// TwinCAT 3 PLC project TRAJ_ADS_SERVER
// ProgramVersion: 3.1.4020.4
// libraries:
//   Tc2_ControllerToolbox, * (Beckhoff Automation GmbH)
//   Tc2_Standard, * (Beckhoff Automation GmbH)
//   Tc2_System, * (Beckhoff Automation GmbH)
//   Tc3_Interfaces, * (Beckhoff Automation GmbH)
//   Tc3_Module, * (Beckhoff Automation GmbH)
// project tree:
//   DUTs/ ROBOT_STATUS.TcDUT (not stored), TRAJECTORY.TcDUT, TRAJ_POINT.TcDUT
//   GVLs/ CONST.TcGVL (not stored)
//   / PlcTask.TcTTO
//   POUs/ MAIN.TcPOU
// real-time tasks:
//   TASK PlcTask: cycle T#1ms, priority 6, ADS port 350
// motion (NC):
//   TASK NC-Task 1 SAF: cycle T#2ms, priority 4, ADS port 501
//   TASK NC-Task 1 SVB: cycle T#10ms, priority 8, ADS port 511
//   AXIS Axis 1 (id 1)
//     OtherSettings: AllowMotionCmdToSlave=true
//     encoder EncType=19
//       EncPara: MaxCount=#xffffffff
//     drive DrvType=16
//       DrvPara: MaxCount=#xffffffff, DriveControlDWord=#x00000100
//         Analog: ScaleFactorActTorque=0.1
//         TimeComp: TaskDelayCycles=1
//     controller CtrType=1
//       CtrPara: PriorControlFactor=1
//         Observer: BandWidth=20
// I/O:
//   DEVICE MY_MOTOR (EtherCAT), AmsNetId 192.168.6.90.3.1
//     Drive 1 (SanyoDenki RS2 EtherCAT) [R ADVANCED MODEL with EtherCAT(P0002813G01)]
// variable links:
//   NC-Task 1 SAF/Axes/Axis 1 <-> MY_MOTOR (EtherCAT)/Drive 1 (SanyoDenki RS2 EtherCAT)
//     Drive/Inputs/In/nDataIn1 <-> Inputs/Following error actualvalue
//     Drive/Inputs/In/nDcOutputTime <-> InfoData/DcOutputShift
//     Drive/Inputs/In/nState1 <-> Inputs/Status word
//     Drive/Inputs/In/nState2 <-> Inputs/Status word @bit 8
//     Drive/Inputs/In/nState4 @bit 1 <-> WcState/InputToggle
//     Drive/Inputs/In/nState4 <-> WcState/WcState
//     Drive/Outputs/Out/nDataOut1 <-> Outputs/Target position
//     Drive/Outputs/Out/nDataOut2 <-> Outputs/Target velocity
//     Enc/Inputs/In/nDataIn3 <-> Inputs/Touch probe position 1 positive value
//     Enc/Inputs/In/nDataIn4 <-> Inputs/Touch probe position 1 negative value
//     Enc/Inputs/In/nDcInputTime <-> InfoData/DcInputShift
//     Enc/Inputs/In/nState4 @bit 1 <-> WcState/InputToggle
//     Enc/Inputs/In/nState4 <-> WcState/WcState
//     Enc/Inputs/In/nState5 <-> Inputs/Touch probe status
//     Enc/Inputs/In/nState6 <-> Inputs/Touch probe status @bit 8
//     Enc/Outputs/Out/nCtrl5 <-> Outputs/Touch probe function
//     Enc/Outputs/Out/nCtrl6 <-> Outputs/Touch probe function @bit 8
//   TRAJ_ADS_SERVER/TRAJ_ADS_SERVER Instance <-> MY_MOTOR (EtherCAT)/Drive 1 (SanyoDenki RS2 EtherCAT)
//     PlcTask Inputs/MAIN.posAct <-> Inputs/Position actual value
//     PlcTask Inputs/MAIN.torAct <-> Inputs/Torque actual value
//     PlcTask Inputs/MAIN.velAct <-> Inputs/Velocity actual value
//     PlcTask Outputs/MAIN.torSet <-> Outputs/Target torque

CONFIGURATION TRAJ_ADS_SERVER
    RESOURCE PLC ON TwinCAT3
        TASK PlcTask(INTERVAL := T#10ms, PRIORITY := 6);
        PROGRAM MAIN WITH PlcTask : MAIN;
    END_RESOURCE
END_CONFIGURATION

// ---- DUTs/TRAJECTORY.TcDUT
TYPE TRAJECTORY :
STRUCT
		size     	  :UINT:=0;                          //轨迹点的数目
		//points        :ARRAY[0..100] OF this_point;      //要执行的一系列轨迹点  
END_STRUCT
END_TYPE

// ---- DUTs/TRAJ_POINT.TcDUT
TYPE TRAJ_POINT :
STRUCT
	joints    : ARRAY [0..6] OF REAL;              //关节的位置数据(7关节)
END_STRUCT
END_TYPE

// ---- POUs/MAIN.TcPOU
PROGRAM MAIN

VAR CONSTANT
	TRAJ_CMD_STOP: 	BYTE :=  0;//停止
	TRAJ_CMD_NEW:   BYTE :=  1;//读入轨迹
	TRAJ_CMD_START: BYTE :=  2;//开始运动
	PULSE_NUM:LREAL:=131072; //编码器脉冲长度
	CYCLE_TICK:BYTE:=1;//周期1us
END_VAR

VAR
	//ADS变量
	traj_cmd                :BYTE:=TRAJ_CMD_STOP; //命令
	traj_size               :UINT:=10;       					//轨迹点的个数
    points        			:ARRAY[0..100] OF TRAJ_POINT;      //要执行的一系列轨迹点 
	joints    : ARRAY [0..6] OF REAL;                  //关节位置数组
	traj_point :TRAJ_POINT;    			   //执行的轨迹点
	last_point :TRAJ_POINT;    			   //执行的轨迹点
	step  :UINT:=0;     		 			//当前轨迹点的步数
	timeStamp     :UDINT:=0; 
	duration      :REAL:=1;
	alpha        :REAL:=0;
	
	//控制程序
	ctrWord   AT%Q*:UINT:=6;//控制模式
	torSet    AT%Q*: INT:=0;
	torAct AT%I*: INT:=0;  //扭矩反馈值(脉冲)
	velAct AT%I*: DINT:=0; //速度反馈值(脉冲)
	posAct AT%I*: DINT:=0; //位置反馈值(脉冲)
	vel: LREAL;             //实际速度
	pos: LREAL;            //实际位置
	
END_VAR

//反馈值
vel:=60*velAct/PULSE_NUM;
pos:=posAct/PULSE_NUM*180;
torSet:=LREAL_TO_INT(50*SIN(0.001*step*0.3));

//根据命令进行操作
CASE traj_cmd OF
TRAJ_CMD_START://CMD:开始执行
			IF step < traj_size AND ctrWord=15 THEN
				duration:=UDINT_TO_REAL(points[step+1].timestamp-points[step].timestamp); //两个轨迹点之间的时间间隔
				alpha:=CYCLE_TICK/duration;//比例系数
				traj_point:=points[step];//获取当前的轨迹点
				//************************EXCUTE MOTION()*********************
				timeStamp:=traj_point.timestamp; //时间
				joints:=traj_point.joints;//关节角度
				step:=step+1;
			ELSE //执行结束时所有将步数清零，命令设置为STOP
				step:=0;
				traj_cmd:=TRAJ_CMD_STOP;
        traj_size：=0
			END_IF
TRAJ_CMD_NEW://CMD：新轨迹
      traj_cmd:=TRAJ_CMD_STOP;
			step:=0;
			//traj_size:=TRAJ.trajectory.size;
			//points:=TRAJ.trajectory.points;

ELSE    //CMD:停止
	torSet:=0;//扭矩置0
END_CASE

METHOD interpolate : BOOL
VAR_INPUT
END_VAR
VAR
	i:BYTE:=0;
END_VAR

//FOR i:=0 TO 6 BY 1 DO
    //this_point.joints[i]:=points[step+1].joints[i]-points[step].joints[i]*alpha;
//END_FOR;
//this_point.timestamp:=points[step+1].timestamp+REAL_TO_UDINT(duration*alpha);
interpolate:=FALSE;
END_METHOD

END_PROGRAM
